FUNCTION_BLOCK fbPIT
VAR_INPUT
	In : REAL;
END_VAR
VAR_OUTPUT
	Pressure : REAL;
	WarningLow : BOOL;
	AlarmLow : BOOL;
	WarningHigh : BOOL;
	AlarmHigh : BOOL;
END_VAR
VAR
	LLLimit : REAL := 10;
	LLimit : REAL := 20;
	HLimit : REAL := 80;
	HHLimit : REAL := 90;
	tDelayTime : TIME := T#0MS;
	tonAL : TON;
	tonWL : TON;
	tonWH : TON;
	tonAH : TON;
END_VAR

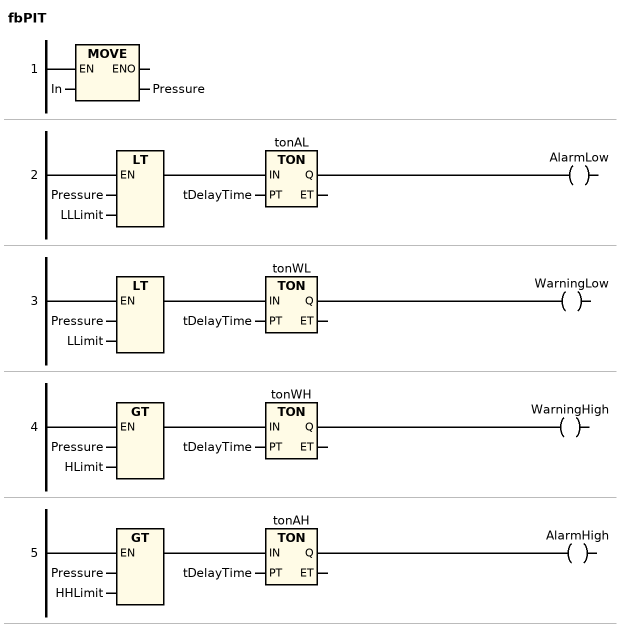
// NETWORK 1
Pressure := In;

// NETWORK 2
tonAL(IN := Pressure < LLLimit, PT := tDelayTime); // TON
AlarmLow := tonAL.Q;

// NETWORK 3
tonWL(IN := Pressure < LLimit, PT := tDelayTime); // TON
WarningLow := tonWL.Q;

// NETWORK 4
tonWH(IN := Pressure > HLimit, PT := tDelayTime); // TON
WarningHigh := tonWH.Q;

// NETWORK 5
tonAH(IN := Pressure > HHLimit, PT := tDelayTime); // TON
AlarmHigh := tonAH.Q;

END_FUNCTION_BLOCK

(* stored: Version 1.1.0.1, ProductVersion 3.1.4022.17
   POU fbPIT: Id {3dab7008-56f3-44dc-883e-dedbc882f6bc}, SpecialFunc None *)
